VAR_GLOBAL
////////////////////////////////////////:	///////////////////////////////////////////////////
/////////////////////////////////////////////////////////////////////////////////////GENERIC/////////////////////////////////////////////////////////////////////////////////////

	bQuitHMI							: BOOL;
	bShutDown							: BOOL;
	stStatusBanner						: ST_StatusBanner;
	nPopUp								: DINT;
	
	bPartPresent						: ARRAY [0..1] OF BOOL;
	
	bRejectPartDialog					: ARRAY [0..2] OF BOOL;
	bOpenRejectDialog					: BOOL;
	bLightsOnOff						: BOOL;
	
	bHMIAlive							: BOOL;
	tonHMIAliveOn						: TON;
	tonHMIAliveOff						: TON;
	bOutHMI								: BOOL;
	bEmptyRejectChuteAcknowledge  		: BOOL;
	bEmptyRejectChute					: BOOL;
	bSavePersistentData					: BOOL;
	
/////////////////////////////////////////////////////////////////////////////////////SYSTEM INFO/////////////////////////////////////////////////////////////////////////////////////

	sSoftwareVersion					: STRING := ' v1.0.0-rc.3';
	sSoftwareDate						: STRING := '03/06/2026';
	sTC3Version							: STRING := ' v3.1.4026.22, Runtime v3.1.4026.22 ';
	sHMIVersion							: STRING := ' 14.13';
	sSystemName							: STRING := 'LT-WH IPX8';
	sProjectID							: STRING := ' TE 11108' ;
	sAplication                     	: STRING ;
	sHMIServer                			: STRING := ' 14.13 ';
	
/////////////////////////////////////////////////////////////////////////////////////MANUAL/////////////////////////////////////////////////////////////////////////////////////

	bEnableManual						: BOOL;
	nMainRegion							: DINT;
	bManualModeOffFlag					: BOOL;
	bManualScreen						: BOOL;
	tonManualMode						: TON;
	bEnableSettings						: BOOL;
	
	stAnimations						: ST_Animations;
	
	bProcessCylinder_Up					: BOOL;
	bProcessCylinderDown				: BOOL;
	bEnableProcessCylinder1				: BOOL;
	
	
	bProcessDoor_Up						: BOOL;
	bProcessDoor_Down					: BOOL;
	
	bSlideNestRight						: BOOL;
	bSlideNestLeft						: BOOL;
	bEnableSildeNest					: BOOL;
	
	bLeaktester1_Start					: BOOL;
	bLeaktester2_Start					: BOOL;
	bLeaktester1_Stop					: BOOL;
	bLeaktester2_Stop					: BOOL;
	bLeaktester1_Reset					: BOOL;
	bLeaktester2_Reset					: BOOL;
	
	
	
	//Probes
	bSetTolerances						: BOOL;
	abPresetProbe						: ARRAY [1..8] OF BOOL;
	bSetCalibrationBlock1				: BOOL;
	bSetCalibrationBlock2				: BOOL;
	bEnableSetCablibrationBlock1		: BOOL;
	bEnableSetCablibrationBlock2		: BOOL;
	bSetDistances						: BOOL;
	(*Renan Added - 30Jun26 - Getting offset from HMI*)
	bSetProbeOffsetNest1				: BOOL;
	(*/Renan Added - 30Jun26 - Getting offset from HMI*)

	(*Renan Added - 06Jul26 - Getting offset from HMI*)
	//Puck Locker
	stPuckLocker 						: ST_PuckLockerHMI;
	(*\Renan Added - 06Jul26 - Getting offset from HMI*)
	
	
	
	
END_VAR

VAR_GLOBAL PERSISTENT
	
	stTimers							: ST_Timers;
	stStatisticsHMI						: ARRAY [0..5] OF ST_StatisticsHMI;	//0: Nest1
																	//1: Nest2
																	//2: Leak Tester 1
																	//3: Leak Tester 2
																	//4: Height Test 1
																	//5: Height Test 2
																	
														
	/////////////////////////////////////////////////////////////////////////////////////SETTINGS/////////////////////////////////////////////////////////////////////////////////////	
	(*Renan Added - 30Jun26 - Getting offset from HMI*)
	anNestOffsetByProbe1         		: ARRAY [1..4] OF REAL;
    anNestOffsetByProbe2         		: ARRAY [1..4] OF REAL;
	(*/Renan Added - 30Jun26 - Getting offset from HMI*)

	(*Renan Added - 06Jul26 - Getting offset from HMI*)
	ePuckLockerMode : E_PuckLockerMode := E_PuckLockerMode.Disabled; //Puck locker state
	bPuckLockerGateEnable 				: BOOL := TRUE;
	bPuckLockerSkipEnable 				: BOOL := FALSE;
	(*\Renan Added - 06Jul26 - Getting offset from HMI*)
	
	
	//TwinSAFE
	
	nAirPressureMaxValue				: UINT;	
	nAirPressureMinValue				: UINT;	
	abMachineDefinition					: ARRAY[1..5] OF  BOOL;
	stTableCycleDataNest1				: ARRAY[0..2000] OF ST_TableCycleData;
	stTableCycleDataNest2				: ARRAY[0..2000] OF ST_TableCycleData;
	
	bNest1Flag							: BOOL;
	bNest2Flag							: BOOL;


	
END_VAR

(* stored: Version 1.1.0.1, ProductVersion 3.1.4026.18
   GVL GVL_HMI: Id {7d424ba3-5d42-48e0-870b-7d749b127bab} *)
